PROGRAM MAIN
VAR
    A:BOOL;
END_VAR

A:=TRUE;//Comment

END_PROGRAM

(* stored: Version 1.1.0.1, ProductVersion 3.1.4024.9
   POU MAIN: Id {a5dab3a8-f5a9-4bfc-aa72-b7ae8c95de15}, SpecialFunc None *)
